// TIA Portal V21 export
DATA_BLOCK "ModeDb_R"   // DB110
{ S7_Optimized_Access := 'FALSE' }
// stored: AutoNumber false
   VAR RETAIN
      ManualMode : "ManualModePara";   // MANUAL MODE
      RunningCycle { S7_SetPoint := 'True'} : "CycleDetails";
      BaseReportPath : String := '/media/simatic/data-storage/Reports/Pdf/';
      FinalReportPath : String;
      ReportId : Int;
      Cycle1 { S7_SetPoint := 'True'} : "ModeParaR";   // PHT
      Cycle2 { S7_SetPoint := 'True'} : "ModeParaR";   // BATCH
      Cycle3 { S7_SetPoint := 'True'} : "ModeParaR";   // SIP
      Cycle4 { S7_SetPoint := 'True'} : "ModeParaR";   // CIP
      Cycle5 { S7_SetPoint := 'True'} : "ModeParaR";   // LOAD CELL CALIBRATION
      ReportName : String[100];
   END_VAR
BEGIN
   RunningCycle.PrintInterval := 30;
END_DATA_BLOCK
